{attribute 'GeneratedUsingTerminal: EK1100-0000-0018'}
{attribute addProperty BoxType "EK1100-0000-0018"}
{attribute addProperty Id "RC40_A2_EK1122RC40_A2_EK1122_EAFADCC873RC40_A3_EK1122RC40_A3_EK1122_E505EE87120RC40_A5_EL1809EL1809_32157CFD20RC40_A6_EL1809EL1809_32157CFD20RC40_A7_EL2809EL2809_2B6483BD19RC40_A8_EL2809EL2809_2B6483BD19RC40_A9_EL2809EL2809_2B6483BD19RC40_1_EndTerminal_EL9010EL9010_D29C20850"}
{attribute addProperty CRC "3105420877"}
{attribute addProperty Size "290"}
{attribute addProperty Name "RC40_1 (EK1100)"}
TYPE RC40_1_EK1100_B918F64D EXTENDS EK1100_1FC0878B :
STRUCT
	{attribute addProperty Name "RC40_A2 (EK1122)"}
	{attribute addProperty PreviousPort "RC40_1 (EK1100) : B"}
	RC40_A2_EK1122 : RC40_A2_EK1122_EAFADCC8;
	{attribute addProperty Name "RC40_A3 (EK1122)"}
	{attribute addProperty PreviousPort "RC40_A2 (EK1122) : C"}
	RC40_A3_EK1122 : RC40_A3_EK1122_E505EE87;
	{attribute addProperty Name "RC40_A5 (EL1809)"}
	{attribute addProperty PreviousPort "RC40_A3 (EK1122) : C"}
	RC40_A5_EL1809 : EL1809_32157CFD;
	{attribute addProperty Name "RC40_A6 (EL1809)"}
	{attribute addProperty PreviousPort "RC40_A5 (EL1809) : B"}
	RC40_A6_EL1809 : EL1809_32157CFD;
	{attribute addProperty Name "RC40_A7 (EL2809)"}
	{attribute addProperty PreviousPort "RC40_A6 (EL1809) : B"}
	RC40_A7_EL2809 : EL2809_2B6483BD;
	{attribute addProperty Name "RC40_A8 (EL2809)"}
	{attribute addProperty PreviousPort "RC40_A7 (EL2809) : B"}
	RC40_A8_EL2809 : EL2809_2B6483BD;
	{attribute addProperty Name "RC40_A9 (EL2809)"}
	{attribute addProperty PreviousPort "RC40_A8 (EL2809) : B"}
	RC40_A9_EL2809 : EL2809_2B6483BD;
	{attribute addProperty Name "RC40_1_EndTerminal (EL9010)"}
	{attribute addProperty PreviousPort "RC40_A9 (EL2809) : B"}
	RC40_1_EndTerminal_EL9010 : EL9010_D29C2085;
END_STRUCT
END_TYPE

(* stored: Version 1.2.0.0, ProductVersion 3.1.4024.11
   DUT RC40_1_EK1100_B918F64D: Id {134cdb16-1e6d-03ef-1d3e-e0370ff26997} *)
